FUNCTION_BLOCK fbCmServo
VAR_IN_OUT
	em : ST_EM;
	cm : ST_CM_SERVO;
END_VAR
VAR
	
END_VAR

END_FUNCTION_BLOCK

(* stored: Version 1.1.0.1, ProductVersion 3.1.4024.12
   POU fbCmServo: Id {151b75ed-c7e6-4971-a72d-672ff46a970f}, SpecialFunc None *)
